PROGRAM MAIN
VAR
	fbLocalSystemTime		:FB_LocalSystemTime;
END_VAR

IF _TaskInfo[GETCURTASKINDEXEX()].FirstCycle THEN
	fbLocalSystemTime(bEnable := TRUE);
END_IF

fbLocalSystemTime();

// This is comment

END_PROGRAM

(* stored: Version 1.1.0.1, ProductVersion 3.1.4024.11
   POU MAIN: Id {013889be-bda3-494b-9de3-9741a4c39185}, SpecialFunc None *)
